// TIA Portal project "Soru8" (V15)

(* hardware
DEVICE "S7-1200 station_1"  S7-1200 Station
   slot 0: "Rack_0"  S7-1200 Rack  Rack  V1.0
   slot 1: "PLC_1"  CPU 1214C DC/DC/DC  6ES7 214-1AG40-0XB0  V4.2
*)

// ===== PLC "PLC_1"  CPU 1214C DC/DC/DC =====

VAR_GLOBAL   // PLC tag table "Default tag table"
   "GirisSensor" AT %I0.0 : Bool;
   "CıkısSensor" AT %I0.1 : Bool;
   "Bos" AT %Q0.0 : Bool;
   "Dolu" AT %Q0.1 : Bool;
   "Deger" AT %MD0 : DWord;
   "GirisBariyer" AT %Q0.2 : Bool;
   "CıkısBariyer" AT %Q0.3 : Bool;
END_VAR

// folder: System blocks/Program resources

DATA_BLOCK "SAyac"   // DB1
{ S7_Optimized_Access := 'TRUE' }
AUTHOR : Simatic
FAMILY : IEC
NAME : UCNTR
VERSION : 1.2
// stored: InstanceOfName IEC_UCOUNTER
"IEC_UCOUNTER"
BEGIN
END_DATA_BLOCK

// folder: (top level)

ORGANIZATION_BLOCK "Main"   // OB1, LAD, ProgramCycle
TITLE = "Main Program Sweep (Cycle)"
{ S7_Optimized_Access := 'TRUE' }
VERSION : 0.1
   VAR_INPUT
      Initial_Call : Bool;   // Initial call of this OB
      Remanence : Bool;   // =True, if remanent data are available
   END_VAR
BEGIN

REGION Network 1: Sayaç bölümü
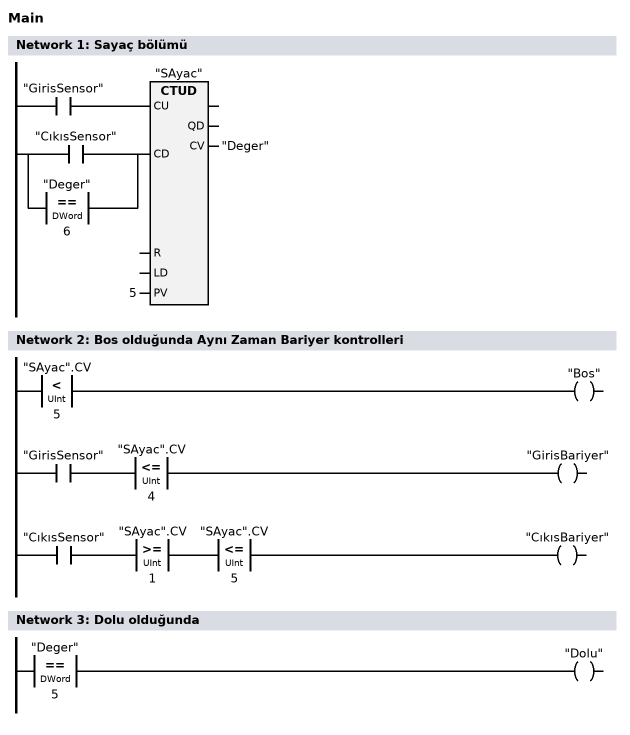
   "SAyac".CTUD(CU := "GirisSensor", CD := "CıkısSensor" OR ("Deger" = 6), PV := 5, CV => "Deger");
END_REGION

REGION Network 2: Bos olduğunda Aynı Zaman Bariyer kontrolleri
   RUNG wire#powerrail
      { S7_Templates := "SrcType := UInt" } LT_Contact(in1 := "SAyac".CV, in2 := 5)
      Coil( "Bos" )
   END_RUNG
   RUNG wire#powerrail
      Contact( "GirisSensor" )
      { S7_Templates := "SrcType := UInt" } LE_Contact(in1 := "SAyac".CV, in2 := 4)
      Coil( "GirisBariyer" )
   END_RUNG
   RUNG wire#powerrail
      Contact( "CıkısSensor" )
      { S7_Templates := "SrcType := UInt" } GE_Contact(in1 := "SAyac".CV, in2 := 1)
      { S7_Templates := "SrcType := UInt" } LE_Contact(in1 := "SAyac".CV, in2 := 5)
      Coil( "CıkısBariyer" )
   END_RUNG
   // the same network as SCL:
   "Bos" := "SAyac".CV < 5;
   "GirisBariyer" := "GirisSensor" AND ("SAyac".CV <= 4);
   "CıkısBariyer" := "CıkısSensor" AND ("SAyac".CV >= 1) AND ("SAyac".CV <= 5);
END_REGION

REGION Network 3: Dolu olduğunda
   RUNG wire#powerrail
      { S7_Templates := "SrcType := DWord" } EQ_Contact(in1 := "Deger", in2 := 5)
      Coil( "Dolu" )
   END_RUNG
   // the same network as SCL:
   "Dolu" := "Deger" = 5;
END_REGION
END_ORGANIZATION_BLOCK